TYPE DUT_stMesOrderItems :
STRUCT
	return_			: DINT;
	OrderReference	: STRING(50);
	OrderItemsJson	: STRING(DB.MAX_STRING_SIZE);
END_STRUCT
END_TYPE

(* stored: Version 1.1.0.1, ProductVersion 3.1.4024.15
   DUT DUT_stMesOrderItems: Id {ba0f42fb-d3a1-4d02-bf34-c7ae4a436d21} *)
